// TIA Portal V16 export
// export: Created 2022-09-01T14:26:55.8686104Z, ExportSetting WithDefaults, DisplayName Totally Integrated Automation Portal, DisplayVersion V16, DisplayName TIA Portal Version Control Interface, DisplayVersion V16, DisplayName TIA Portal Openness, DisplayVersion V16, DisplayName STEP 7 Professional, DisplayVersion V16, DisplayName STEP 7 Safety, DisplayVersion V16, DisplayName WinCC Advanced, DisplayVersion V16
FUNCTION "Ciclo_Limpeza" : Void   // FC1, LAD
TITLE = Ciclo de lavagem e enxaguamento
{ S7_Optimized_Access := 'TRUE' }
VERSION : 0.1
// stored: AutoNumber true, IsIECCheckEnabled false, SetENOAutomatically false, UDAEnableTagReadback false
   VAR_TEMP   // added for the SCL form of the ladder/FBD networks
      _w1 : Bool;
      _w2 : Bool;
      _w3 : Bool;
   END_VAR
BEGIN

REGION Network 1: Etapa 1 (Início)
   // Início com EV's na posição de filtração. As bombas podem estar ligadas ou não, conforme a posição do switch 4
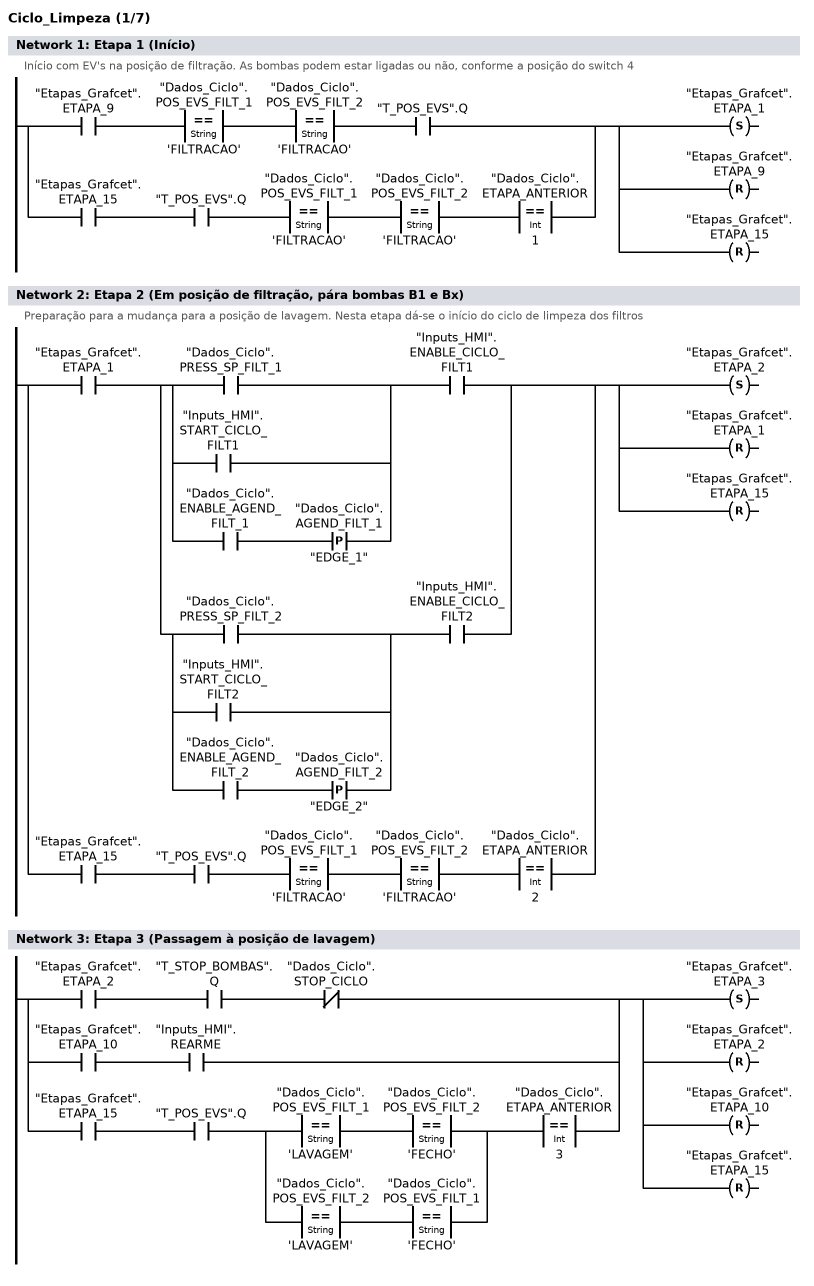
   RUNG wire#powerrail
      Contact( "Etapas_Grafcet".ETAPA_9 )
      { S7_Templates := "SrcType := String" } EQ_Contact(in1 := "Dados_Ciclo".POS_EVS_FILT_1, in2 := 'FILTRACAO')
      { S7_Templates := "SrcType := String" } EQ_Contact(in1 := "Dados_Ciclo".POS_EVS_FILT_2, in2 := 'FILTRACAO')
      Contact( "T_POS_EVS".Q )
      wire#w1
      S_Coil( "Etapas_Grafcet".ETAPA_1 )
   END_RUNG
   RUNG wire#powerrail
      Contact( "Etapas_Grafcet".ETAPA_15 )
      Contact( "T_POS_EVS".Q )
      { S7_Templates := "SrcType := String" } EQ_Contact(in1 := "Dados_Ciclo".POS_EVS_FILT_1, in2 := 'FILTRACAO')
      { S7_Templates := "SrcType := String" } EQ_Contact(in1 := "Dados_Ciclo".POS_EVS_FILT_2, in2 := 'FILTRACAO')
      { S7_Templates := "SrcType := Int" } EQ_Contact(in1 := "Dados_Ciclo".ETAPA_ANTERIOR, in2 := 1)
   END_RUNG wire#w1
   RUNG wire#w1
      R_Coil( "Etapas_Grafcet".ETAPA_9 )
   END_RUNG
   RUNG wire#w1
      R_Coil( "Etapas_Grafcet".ETAPA_15 )
   END_RUNG
   // the same network as SCL:
   IF ("Etapas_Grafcet".ETAPA_9 AND ("Dados_Ciclo".POS_EVS_FILT_1 = 'FILTRACAO') AND ("Dados_Ciclo".POS_EVS_FILT_2 = 'FILTRACAO') AND "T_POS_EVS".Q) OR ("Etapas_Grafcet".ETAPA_15 AND "T_POS_EVS".Q AND ("Dados_Ciclo".POS_EVS_FILT_1 = 'FILTRACAO') AND ("Dados_Ciclo".POS_EVS_FILT_2 = 'FILTRACAO') AND ("Dados_Ciclo".ETAPA_ANTERIOR = 1)) THEN
       "Etapas_Grafcet".ETAPA_1 := TRUE;
   END_IF;
   #_w1 := ("Etapas_Grafcet".ETAPA_9 AND ("Dados_Ciclo".POS_EVS_FILT_1 = 'FILTRACAO') AND ("Dados_Ciclo".POS_EVS_FILT_2 = 'FILTRACAO') AND "T_POS_EVS".Q) OR ("Etapas_Grafcet".ETAPA_15 AND "T_POS_EVS".Q AND ("Dados_Ciclo".POS_EVS_FILT_1 = 'FILTRACAO') AND ("Dados_Ciclo".POS_EVS_FILT_2 = 'FILTRACAO') AND ("Dados_Ciclo".ETAPA_ANTERIOR = 1));
   IF #_w1 THEN
       "Etapas_Grafcet".ETAPA_9 := FALSE;
       "Etapas_Grafcet".ETAPA_15 := FALSE;
   END_IF;
END_REGION

REGION Network 2: Etapa 2 (Em posição de filtração, pára bombas B1 e Bx)
   // Preparação para a mudança para a posição de lavagem. Nesta etapa dá-se o início do ciclo de limpeza dos filtros
   RUNG wire#powerrail
      Contact( "Etapas_Grafcet".ETAPA_1 )
      wire#w1
      Contact( "Dados_Ciclo".PRESS_SP_FILT_1 )
      wire#w2
      Contact( "Inputs_HMI".ENABLE_CICLO_FILT1 )
      wire#w3
      S_Coil( "Etapas_Grafcet".ETAPA_2 )
   END_RUNG
   RUNG wire#w1
      Contact( "Inputs_HMI".START_CICLO_FILT1 )
   END_RUNG wire#w2
   RUNG wire#w1
      Contact( "Dados_Ciclo".ENABLE_AGEND_FILT_1 )
      P_Contact(operand := "Dados_Ciclo".AGEND_FILT_1, bit := "EDGE_1")
   END_RUNG wire#w2
   RUNG wire#w1
      Contact( "Dados_Ciclo".PRESS_SP_FILT_2 )
      wire#w4
      Contact( "Inputs_HMI".ENABLE_CICLO_FILT2 )
   END_RUNG wire#w3
   RUNG wire#w1
      Contact( "Inputs_HMI".START_CICLO_FILT2 )
   END_RUNG wire#w4
   RUNG wire#w1
      Contact( "Dados_Ciclo".ENABLE_AGEND_FILT_2 )
      P_Contact(operand := "Dados_Ciclo".AGEND_FILT_2, bit := "EDGE_2")
   END_RUNG wire#w4
   RUNG wire#powerrail
      Contact( "Etapas_Grafcet".ETAPA_15 )
      Contact( "T_POS_EVS".Q )
      { S7_Templates := "SrcType := String" } EQ_Contact(in1 := "Dados_Ciclo".POS_EVS_FILT_1, in2 := 'FILTRACAO')
      { S7_Templates := "SrcType := String" } EQ_Contact(in1 := "Dados_Ciclo".POS_EVS_FILT_2, in2 := 'FILTRACAO')
      { S7_Templates := "SrcType := Int" } EQ_Contact(in1 := "Dados_Ciclo".ETAPA_ANTERIOR, in2 := 2)
   END_RUNG wire#w3
   RUNG wire#w3
      R_Coil( "Etapas_Grafcet".ETAPA_1 )
   END_RUNG
   RUNG wire#w3
      R_Coil( "Etapas_Grafcet".ETAPA_15 )
   END_RUNG
   // the same network as SCL:
   #_w1 := "Etapas_Grafcet".ETAPA_1 AND "Dados_Ciclo".ENABLE_AGEND_FILT_1 AND "Dados_Ciclo".AGEND_FILT_1 AND NOT "EDGE_1";   // rising edge of "Dados_Ciclo".AGEND_FILT_1
   "EDGE_1" := "Dados_Ciclo".AGEND_FILT_1;
   #_w2 := "Etapas_Grafcet".ETAPA_1 AND "Dados_Ciclo".ENABLE_AGEND_FILT_2 AND "Dados_Ciclo".AGEND_FILT_2 AND NOT "EDGE_2";   // rising edge of "Dados_Ciclo".AGEND_FILT_2
   "EDGE_2" := "Dados_Ciclo".AGEND_FILT_2;
   IF ((("Etapas_Grafcet".ETAPA_1 AND ("Dados_Ciclo".PRESS_SP_FILT_1 OR "Inputs_HMI".START_CICLO_FILT1)) OR #_w1) AND "Inputs_HMI".ENABLE_CICLO_FILT1) OR ((("Etapas_Grafcet".ETAPA_1 AND ("Dados_Ciclo".PRESS_SP_FILT_2 OR "Inputs_HMI".START_CICLO_FILT2)) OR #_w2) AND "Inputs_HMI".ENABLE_CICLO_FILT2) OR ("Etapas_Grafcet".ETAPA_15 AND "T_POS_EVS".Q AND ("Dados_Ciclo".POS_EVS_FILT_1 = 'FILTRACAO') AND ("Dados_Ciclo".POS_EVS_FILT_2 = 'FILTRACAO') AND ("Dados_Ciclo".ETAPA_ANTERIOR = 2)) THEN
       "Etapas_Grafcet".ETAPA_2 := TRUE;
   END_IF;
   #_w3 := ((("Etapas_Grafcet".ETAPA_1 AND ("Dados_Ciclo".PRESS_SP_FILT_1 OR "Inputs_HMI".START_CICLO_FILT1)) OR #_w1) AND "Inputs_HMI".ENABLE_CICLO_FILT1) OR ((("Etapas_Grafcet".ETAPA_1 AND ("Dados_Ciclo".PRESS_SP_FILT_2 OR "Inputs_HMI".START_CICLO_FILT2)) OR #_w2) AND "Inputs_HMI".ENABLE_CICLO_FILT2) OR ("Etapas_Grafcet".ETAPA_15 AND "T_POS_EVS".Q AND ("Dados_Ciclo".POS_EVS_FILT_1 = 'FILTRACAO') AND ("Dados_Ciclo".POS_EVS_FILT_2 = 'FILTRACAO') AND ("Dados_Ciclo".ETAPA_ANTERIOR = 2));
   IF #_w3 THEN
       "Etapas_Grafcet".ETAPA_1 := FALSE;
       "Etapas_Grafcet".ETAPA_15 := FALSE;
   END_IF;
END_REGION

REGION Network 3: Etapa 3 (Passagem à posição de lavagem)
   RUNG wire#powerrail
      Contact( "Etapas_Grafcet".ETAPA_2 )
      Contact( "T_STOP_BOMBAS".Q )
      I_Contact( "Dados_Ciclo".STOP_CICLO )
      wire#w1
      S_Coil( "Etapas_Grafcet".ETAPA_3 )
   END_RUNG
   RUNG wire#powerrail
      Contact( "Etapas_Grafcet".ETAPA_10 )
      Contact( "Inputs_HMI".REARME )
   END_RUNG wire#w1
   RUNG wire#powerrail
      Contact( "Etapas_Grafcet".ETAPA_15 )
      Contact( "T_POS_EVS".Q )
      wire#w2
      { S7_Templates := "SrcType := String" } EQ_Contact(in1 := "Dados_Ciclo".POS_EVS_FILT_1, in2 := 'LAVAGEM')
      { S7_Templates := "SrcType := String" } EQ_Contact(in1 := "Dados_Ciclo".POS_EVS_FILT_2, in2 := 'FECHO')
      wire#w3
      { S7_Templates := "SrcType := Int" } EQ_Contact(in1 := "Dados_Ciclo".ETAPA_ANTERIOR, in2 := 3)
   END_RUNG wire#w1
   RUNG wire#w2
      { S7_Templates := "SrcType := String" } EQ_Contact(in1 := "Dados_Ciclo".POS_EVS_FILT_2, in2 := 'LAVAGEM')
      { S7_Templates := "SrcType := String" } EQ_Contact(in1 := "Dados_Ciclo".POS_EVS_FILT_1, in2 := 'FECHO')
   END_RUNG wire#w3
   RUNG wire#w1
      R_Coil( "Etapas_Grafcet".ETAPA_2 )
   END_RUNG
   RUNG wire#w1
      R_Coil( "Etapas_Grafcet".ETAPA_10 )
   END_RUNG
   RUNG wire#w1
      R_Coil( "Etapas_Grafcet".ETAPA_15 )
   END_RUNG
   // the same network as SCL:
   IF ("Etapas_Grafcet".ETAPA_2 AND "T_STOP_BOMBAS".Q AND NOT "Dados_Ciclo".STOP_CICLO) OR ("Etapas_Grafcet".ETAPA_10 AND "Inputs_HMI".REARME) OR ("Etapas_Grafcet".ETAPA_15 AND "T_POS_EVS".Q AND ((("Dados_Ciclo".POS_EVS_FILT_1 = 'LAVAGEM') AND ("Dados_Ciclo".POS_EVS_FILT_2 = 'FECHO')) OR (("Dados_Ciclo".POS_EVS_FILT_2 = 'LAVAGEM') AND ("Dados_Ciclo".POS_EVS_FILT_1 = 'FECHO'))) AND ("Dados_Ciclo".ETAPA_ANTERIOR = 3)) THEN
       "Etapas_Grafcet".ETAPA_3 := TRUE;
   END_IF;
   #_w1 := ("Etapas_Grafcet".ETAPA_2 AND "T_STOP_BOMBAS".Q AND NOT "Dados_Ciclo".STOP_CICLO) OR ("Etapas_Grafcet".ETAPA_10 AND "Inputs_HMI".REARME) OR ("Etapas_Grafcet".ETAPA_15 AND "T_POS_EVS".Q AND ((("Dados_Ciclo".POS_EVS_FILT_1 = 'LAVAGEM') AND ("Dados_Ciclo".POS_EVS_FILT_2 = 'FECHO')) OR (("Dados_Ciclo".POS_EVS_FILT_2 = 'LAVAGEM') AND ("Dados_Ciclo".POS_EVS_FILT_1 = 'FECHO'))) AND ("Dados_Ciclo".ETAPA_ANTERIOR = 3));
   IF #_w1 THEN
       "Etapas_Grafcet".ETAPA_2 := FALSE;
       "Etapas_Grafcet".ETAPA_10 := FALSE;
       "Etapas_Grafcet".ETAPA_15 := FALSE;
   END_IF;
END_REGION

REGION Network 4: Etapa 4 (Em lavagem, B1 e BX ligadas)
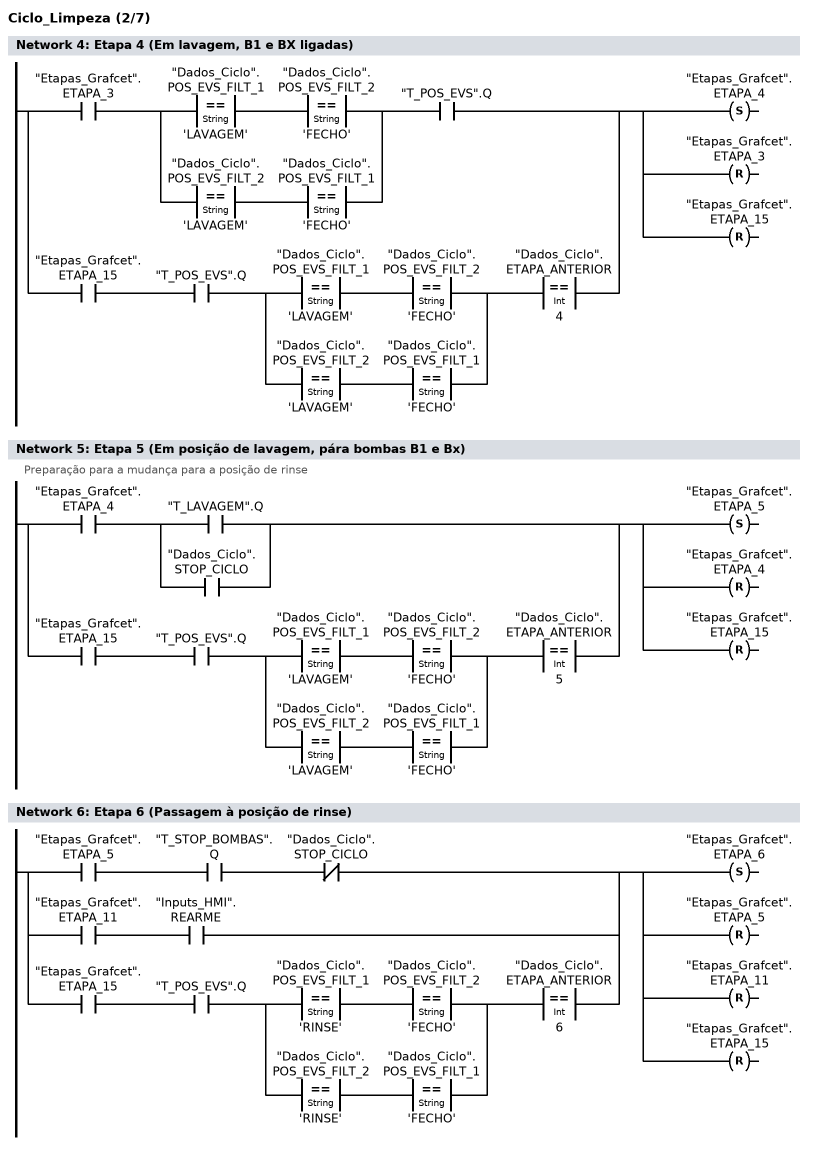
   RUNG wire#powerrail
      Contact( "Etapas_Grafcet".ETAPA_3 )
      wire#w1
      { S7_Templates := "SrcType := String" } EQ_Contact(in1 := "Dados_Ciclo".POS_EVS_FILT_1, in2 := 'LAVAGEM')
      { S7_Templates := "SrcType := String" } EQ_Contact(in1 := "Dados_Ciclo".POS_EVS_FILT_2, in2 := 'FECHO')
      wire#w2
      Contact( "T_POS_EVS".Q )
      wire#w3
      S_Coil( "Etapas_Grafcet".ETAPA_4 )
   END_RUNG
   RUNG wire#w1
      { S7_Templates := "SrcType := String" } EQ_Contact(in1 := "Dados_Ciclo".POS_EVS_FILT_2, in2 := 'LAVAGEM')
      { S7_Templates := "SrcType := String" } EQ_Contact(in1 := "Dados_Ciclo".POS_EVS_FILT_1, in2 := 'FECHO')
   END_RUNG wire#w2
   RUNG wire#powerrail
      Contact( "Etapas_Grafcet".ETAPA_15 )
      Contact( "T_POS_EVS".Q )
      wire#w4
      { S7_Templates := "SrcType := String" } EQ_Contact(in1 := "Dados_Ciclo".POS_EVS_FILT_1, in2 := 'LAVAGEM')
      { S7_Templates := "SrcType := String" } EQ_Contact(in1 := "Dados_Ciclo".POS_EVS_FILT_2, in2 := 'FECHO')
      wire#w5
      { S7_Templates := "SrcType := Int" } EQ_Contact(in1 := "Dados_Ciclo".ETAPA_ANTERIOR, in2 := 4)
   END_RUNG wire#w3
   RUNG wire#w4
      { S7_Templates := "SrcType := String" } EQ_Contact(in1 := "Dados_Ciclo".POS_EVS_FILT_2, in2 := 'LAVAGEM')
      { S7_Templates := "SrcType := String" } EQ_Contact(in1 := "Dados_Ciclo".POS_EVS_FILT_1, in2 := 'FECHO')
   END_RUNG wire#w5
   RUNG wire#w3
      R_Coil( "Etapas_Grafcet".ETAPA_3 )
   END_RUNG
   RUNG wire#w3
      R_Coil( "Etapas_Grafcet".ETAPA_15 )
   END_RUNG
   // the same network as SCL:
   IF ("Etapas_Grafcet".ETAPA_3 AND ((("Dados_Ciclo".POS_EVS_FILT_1 = 'LAVAGEM') AND ("Dados_Ciclo".POS_EVS_FILT_2 = 'FECHO')) OR (("Dados_Ciclo".POS_EVS_FILT_2 = 'LAVAGEM') AND ("Dados_Ciclo".POS_EVS_FILT_1 = 'FECHO'))) AND "T_POS_EVS".Q) OR ("Etapas_Grafcet".ETAPA_15 AND "T_POS_EVS".Q AND ((("Dados_Ciclo".POS_EVS_FILT_1 = 'LAVAGEM') AND ("Dados_Ciclo".POS_EVS_FILT_2 = 'FECHO')) OR (("Dados_Ciclo".POS_EVS_FILT_2 = 'LAVAGEM') AND ("Dados_Ciclo".POS_EVS_FILT_1 = 'FECHO'))) AND ("Dados_Ciclo".ETAPA_ANTERIOR = 4)) THEN
       "Etapas_Grafcet".ETAPA_4 := TRUE;
   END_IF;
   #_w1 := ("Etapas_Grafcet".ETAPA_3 AND ((("Dados_Ciclo".POS_EVS_FILT_1 = 'LAVAGEM') AND ("Dados_Ciclo".POS_EVS_FILT_2 = 'FECHO')) OR (("Dados_Ciclo".POS_EVS_FILT_2 = 'LAVAGEM') AND ("Dados_Ciclo".POS_EVS_FILT_1 = 'FECHO'))) AND "T_POS_EVS".Q) OR ("Etapas_Grafcet".ETAPA_15 AND "T_POS_EVS".Q AND ((("Dados_Ciclo".POS_EVS_FILT_1 = 'LAVAGEM') AND ("Dados_Ciclo".POS_EVS_FILT_2 = 'FECHO')) OR (("Dados_Ciclo".POS_EVS_FILT_2 = 'LAVAGEM') AND ("Dados_Ciclo".POS_EVS_FILT_1 = 'FECHO'))) AND ("Dados_Ciclo".ETAPA_ANTERIOR = 4));
   IF #_w1 THEN
       "Etapas_Grafcet".ETAPA_3 := FALSE;
       "Etapas_Grafcet".ETAPA_15 := FALSE;
   END_IF;
END_REGION

REGION Network 5: Etapa 5 (Em posição de lavagem, pára bombas B1 e Bx)
   // Preparação para a mudança para a posição de rinse
   RUNG wire#powerrail
      Contact( "Etapas_Grafcet".ETAPA_4 )
      wire#w1
      Contact( "T_LAVAGEM".Q )
      wire#w2
      S_Coil( "Etapas_Grafcet".ETAPA_5 )
   END_RUNG
   RUNG wire#w1
      Contact( "Dados_Ciclo".STOP_CICLO )
   END_RUNG wire#w2
   RUNG wire#powerrail
      Contact( "Etapas_Grafcet".ETAPA_15 )
      Contact( "T_POS_EVS".Q )
      wire#w3
      { S7_Templates := "SrcType := String" } EQ_Contact(in1 := "Dados_Ciclo".POS_EVS_FILT_1, in2 := 'LAVAGEM')
      { S7_Templates := "SrcType := String" } EQ_Contact(in1 := "Dados_Ciclo".POS_EVS_FILT_2, in2 := 'FECHO')
      wire#w4
      { S7_Templates := "SrcType := Int" } EQ_Contact(in1 := "Dados_Ciclo".ETAPA_ANTERIOR, in2 := 5)
   END_RUNG wire#w2
   RUNG wire#w3
      { S7_Templates := "SrcType := String" } EQ_Contact(in1 := "Dados_Ciclo".POS_EVS_FILT_2, in2 := 'LAVAGEM')
      { S7_Templates := "SrcType := String" } EQ_Contact(in1 := "Dados_Ciclo".POS_EVS_FILT_1, in2 := 'FECHO')
   END_RUNG wire#w4
   RUNG wire#w2
      R_Coil( "Etapas_Grafcet".ETAPA_4 )
   END_RUNG
   RUNG wire#w2
      R_Coil( "Etapas_Grafcet".ETAPA_15 )
   END_RUNG
   // the same network as SCL:
   IF ("Etapas_Grafcet".ETAPA_4 AND ("T_LAVAGEM".Q OR "Dados_Ciclo".STOP_CICLO)) OR ("Etapas_Grafcet".ETAPA_15 AND "T_POS_EVS".Q AND ((("Dados_Ciclo".POS_EVS_FILT_1 = 'LAVAGEM') AND ("Dados_Ciclo".POS_EVS_FILT_2 = 'FECHO')) OR (("Dados_Ciclo".POS_EVS_FILT_2 = 'LAVAGEM') AND ("Dados_Ciclo".POS_EVS_FILT_1 = 'FECHO'))) AND ("Dados_Ciclo".ETAPA_ANTERIOR = 5)) THEN
       "Etapas_Grafcet".ETAPA_5 := TRUE;
   END_IF;
   #_w1 := ("Etapas_Grafcet".ETAPA_4 AND ("T_LAVAGEM".Q OR "Dados_Ciclo".STOP_CICLO)) OR ("Etapas_Grafcet".ETAPA_15 AND "T_POS_EVS".Q AND ((("Dados_Ciclo".POS_EVS_FILT_1 = 'LAVAGEM') AND ("Dados_Ciclo".POS_EVS_FILT_2 = 'FECHO')) OR (("Dados_Ciclo".POS_EVS_FILT_2 = 'LAVAGEM') AND ("Dados_Ciclo".POS_EVS_FILT_1 = 'FECHO'))) AND ("Dados_Ciclo".ETAPA_ANTERIOR = 5));
   IF #_w1 THEN
       "Etapas_Grafcet".ETAPA_4 := FALSE;
       "Etapas_Grafcet".ETAPA_15 := FALSE;
   END_IF;
END_REGION

REGION Network 6: Etapa 6 (Passagem à posição de rinse)
   RUNG wire#powerrail
      Contact( "Etapas_Grafcet".ETAPA_5 )
      Contact( "T_STOP_BOMBAS".Q )
      I_Contact( "Dados_Ciclo".STOP_CICLO )
      wire#w1
      S_Coil( "Etapas_Grafcet".ETAPA_6 )
   END_RUNG
   RUNG wire#powerrail
      Contact( "Etapas_Grafcet".ETAPA_11 )
      Contact( "Inputs_HMI".REARME )
   END_RUNG wire#w1
   RUNG wire#powerrail
      Contact( "Etapas_Grafcet".ETAPA_15 )
      Contact( "T_POS_EVS".Q )
      wire#w2
      { S7_Templates := "SrcType := String" } EQ_Contact(in1 := "Dados_Ciclo".POS_EVS_FILT_1, in2 := 'RINSE')
      { S7_Templates := "SrcType := String" } EQ_Contact(in1 := "Dados_Ciclo".POS_EVS_FILT_2, in2 := 'FECHO')
      wire#w3
      { S7_Templates := "SrcType := Int" } EQ_Contact(in1 := "Dados_Ciclo".ETAPA_ANTERIOR, in2 := 6)
   END_RUNG wire#w1
   RUNG wire#w2
      { S7_Templates := "SrcType := String" } EQ_Contact(in1 := "Dados_Ciclo".POS_EVS_FILT_2, in2 := 'RINSE')
      { S7_Templates := "SrcType := String" } EQ_Contact(in1 := "Dados_Ciclo".POS_EVS_FILT_1, in2 := 'FECHO')
   END_RUNG wire#w3
   RUNG wire#w1
      R_Coil( "Etapas_Grafcet".ETAPA_5 )
   END_RUNG
   RUNG wire#w1
      R_Coil( "Etapas_Grafcet".ETAPA_11 )
   END_RUNG
   RUNG wire#w1
      R_Coil( "Etapas_Grafcet".ETAPA_15 )
   END_RUNG
   // the same network as SCL:
   IF ("Etapas_Grafcet".ETAPA_5 AND "T_STOP_BOMBAS".Q AND NOT "Dados_Ciclo".STOP_CICLO) OR ("Etapas_Grafcet".ETAPA_11 AND "Inputs_HMI".REARME) OR ("Etapas_Grafcet".ETAPA_15 AND "T_POS_EVS".Q AND ((("Dados_Ciclo".POS_EVS_FILT_1 = 'RINSE') AND ("Dados_Ciclo".POS_EVS_FILT_2 = 'FECHO')) OR (("Dados_Ciclo".POS_EVS_FILT_2 = 'RINSE') AND ("Dados_Ciclo".POS_EVS_FILT_1 = 'FECHO'))) AND ("Dados_Ciclo".ETAPA_ANTERIOR = 6)) THEN
       "Etapas_Grafcet".ETAPA_6 := TRUE;
   END_IF;
   #_w1 := ("Etapas_Grafcet".ETAPA_5 AND "T_STOP_BOMBAS".Q AND NOT "Dados_Ciclo".STOP_CICLO) OR ("Etapas_Grafcet".ETAPA_11 AND "Inputs_HMI".REARME) OR ("Etapas_Grafcet".ETAPA_15 AND "T_POS_EVS".Q AND ((("Dados_Ciclo".POS_EVS_FILT_1 = 'RINSE') AND ("Dados_Ciclo".POS_EVS_FILT_2 = 'FECHO')) OR (("Dados_Ciclo".POS_EVS_FILT_2 = 'RINSE') AND ("Dados_Ciclo".POS_EVS_FILT_1 = 'FECHO'))) AND ("Dados_Ciclo".ETAPA_ANTERIOR = 6));
   IF #_w1 THEN
       "Etapas_Grafcet".ETAPA_5 := FALSE;
       "Etapas_Grafcet".ETAPA_11 := FALSE;
       "Etapas_Grafcet".ETAPA_15 := FALSE;
   END_IF;
END_REGION

REGION Network 7: Etapa 7 (Em rinse, B1 ligada)
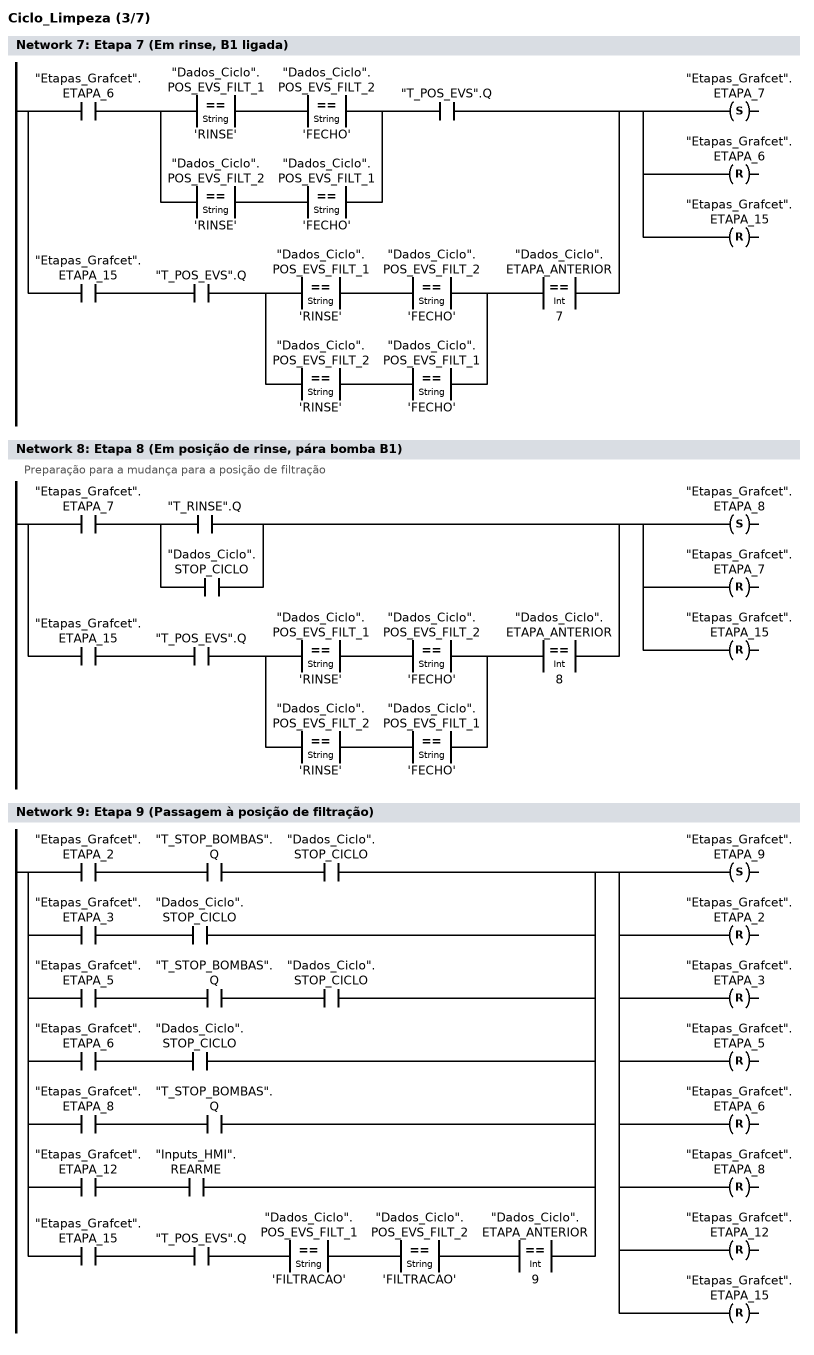
   RUNG wire#powerrail
      Contact( "Etapas_Grafcet".ETAPA_6 )
      wire#w1
      { S7_Templates := "SrcType := String" } EQ_Contact(in1 := "Dados_Ciclo".POS_EVS_FILT_1, in2 := 'RINSE')
      { S7_Templates := "SrcType := String" } EQ_Contact(in1 := "Dados_Ciclo".POS_EVS_FILT_2, in2 := 'FECHO')
      wire#w2
      Contact( "T_POS_EVS".Q )
      wire#w3
      S_Coil( "Etapas_Grafcet".ETAPA_7 )
   END_RUNG
   RUNG wire#w1
      { S7_Templates := "SrcType := String" } EQ_Contact(in1 := "Dados_Ciclo".POS_EVS_FILT_2, in2 := 'RINSE')
      { S7_Templates := "SrcType := String" } EQ_Contact(in1 := "Dados_Ciclo".POS_EVS_FILT_1, in2 := 'FECHO')
   END_RUNG wire#w2
   RUNG wire#powerrail
      Contact( "Etapas_Grafcet".ETAPA_15 )
      Contact( "T_POS_EVS".Q )
      wire#w4
      { S7_Templates := "SrcType := String" } EQ_Contact(in1 := "Dados_Ciclo".POS_EVS_FILT_1, in2 := 'RINSE')
      { S7_Templates := "SrcType := String" } EQ_Contact(in1 := "Dados_Ciclo".POS_EVS_FILT_2, in2 := 'FECHO')
      wire#w5
      { S7_Templates := "SrcType := Int" } EQ_Contact(in1 := "Dados_Ciclo".ETAPA_ANTERIOR, in2 := 7)
   END_RUNG wire#w3
   RUNG wire#w4
      { S7_Templates := "SrcType := String" } EQ_Contact(in1 := "Dados_Ciclo".POS_EVS_FILT_2, in2 := 'RINSE')
      { S7_Templates := "SrcType := String" } EQ_Contact(in1 := "Dados_Ciclo".POS_EVS_FILT_1, in2 := 'FECHO')
   END_RUNG wire#w5
   RUNG wire#w3
      R_Coil( "Etapas_Grafcet".ETAPA_6 )
   END_RUNG
   RUNG wire#w3
      R_Coil( "Etapas_Grafcet".ETAPA_15 )
   END_RUNG
   // the same network as SCL:
   IF ("Etapas_Grafcet".ETAPA_6 AND ((("Dados_Ciclo".POS_EVS_FILT_1 = 'RINSE') AND ("Dados_Ciclo".POS_EVS_FILT_2 = 'FECHO')) OR (("Dados_Ciclo".POS_EVS_FILT_2 = 'RINSE') AND ("Dados_Ciclo".POS_EVS_FILT_1 = 'FECHO'))) AND "T_POS_EVS".Q) OR ("Etapas_Grafcet".ETAPA_15 AND "T_POS_EVS".Q AND ((("Dados_Ciclo".POS_EVS_FILT_1 = 'RINSE') AND ("Dados_Ciclo".POS_EVS_FILT_2 = 'FECHO')) OR (("Dados_Ciclo".POS_EVS_FILT_2 = 'RINSE') AND ("Dados_Ciclo".POS_EVS_FILT_1 = 'FECHO'))) AND ("Dados_Ciclo".ETAPA_ANTERIOR = 7)) THEN
       "Etapas_Grafcet".ETAPA_7 := TRUE;
   END_IF;
   #_w1 := ("Etapas_Grafcet".ETAPA_6 AND ((("Dados_Ciclo".POS_EVS_FILT_1 = 'RINSE') AND ("Dados_Ciclo".POS_EVS_FILT_2 = 'FECHO')) OR (("Dados_Ciclo".POS_EVS_FILT_2 = 'RINSE') AND ("Dados_Ciclo".POS_EVS_FILT_1 = 'FECHO'))) AND "T_POS_EVS".Q) OR ("Etapas_Grafcet".ETAPA_15 AND "T_POS_EVS".Q AND ((("Dados_Ciclo".POS_EVS_FILT_1 = 'RINSE') AND ("Dados_Ciclo".POS_EVS_FILT_2 = 'FECHO')) OR (("Dados_Ciclo".POS_EVS_FILT_2 = 'RINSE') AND ("Dados_Ciclo".POS_EVS_FILT_1 = 'FECHO'))) AND ("Dados_Ciclo".ETAPA_ANTERIOR = 7));
   IF #_w1 THEN
       "Etapas_Grafcet".ETAPA_6 := FALSE;
       "Etapas_Grafcet".ETAPA_15 := FALSE;
   END_IF;
END_REGION

REGION Network 8: Etapa 8 (Em posição de rinse, pára bomba B1)
   // Preparação para a mudança para a posição de filtração
   RUNG wire#powerrail
      Contact( "Etapas_Grafcet".ETAPA_7 )
      wire#w1
      Contact( "T_RINSE".Q )
      wire#w2
      S_Coil( "Etapas_Grafcet".ETAPA_8 )
   END_RUNG
   RUNG wire#w1
      Contact( "Dados_Ciclo".STOP_CICLO )
   END_RUNG wire#w2
   RUNG wire#powerrail
      Contact( "Etapas_Grafcet".ETAPA_15 )
      Contact( "T_POS_EVS".Q )
      wire#w3
      { S7_Templates := "SrcType := String" } EQ_Contact(in1 := "Dados_Ciclo".POS_EVS_FILT_1, in2 := 'RINSE')
      { S7_Templates := "SrcType := String" } EQ_Contact(in1 := "Dados_Ciclo".POS_EVS_FILT_2, in2 := 'FECHO')
      wire#w4
      { S7_Templates := "SrcType := Int" } EQ_Contact(in1 := "Dados_Ciclo".ETAPA_ANTERIOR, in2 := 8)
   END_RUNG wire#w2
   RUNG wire#w3
      { S7_Templates := "SrcType := String" } EQ_Contact(in1 := "Dados_Ciclo".POS_EVS_FILT_2, in2 := 'RINSE')
      { S7_Templates := "SrcType := String" } EQ_Contact(in1 := "Dados_Ciclo".POS_EVS_FILT_1, in2 := 'FECHO')
   END_RUNG wire#w4
   RUNG wire#w2
      R_Coil( "Etapas_Grafcet".ETAPA_7 )
   END_RUNG
   RUNG wire#w2
      R_Coil( "Etapas_Grafcet".ETAPA_15 )
   END_RUNG
   // the same network as SCL:
   IF ("Etapas_Grafcet".ETAPA_7 AND ("T_RINSE".Q OR "Dados_Ciclo".STOP_CICLO)) OR ("Etapas_Grafcet".ETAPA_15 AND "T_POS_EVS".Q AND ((("Dados_Ciclo".POS_EVS_FILT_1 = 'RINSE') AND ("Dados_Ciclo".POS_EVS_FILT_2 = 'FECHO')) OR (("Dados_Ciclo".POS_EVS_FILT_2 = 'RINSE') AND ("Dados_Ciclo".POS_EVS_FILT_1 = 'FECHO'))) AND ("Dados_Ciclo".ETAPA_ANTERIOR = 8)) THEN
       "Etapas_Grafcet".ETAPA_8 := TRUE;
   END_IF;
   #_w1 := ("Etapas_Grafcet".ETAPA_7 AND ("T_RINSE".Q OR "Dados_Ciclo".STOP_CICLO)) OR ("Etapas_Grafcet".ETAPA_15 AND "T_POS_EVS".Q AND ((("Dados_Ciclo".POS_EVS_FILT_1 = 'RINSE') AND ("Dados_Ciclo".POS_EVS_FILT_2 = 'FECHO')) OR (("Dados_Ciclo".POS_EVS_FILT_2 = 'RINSE') AND ("Dados_Ciclo".POS_EVS_FILT_1 = 'FECHO'))) AND ("Dados_Ciclo".ETAPA_ANTERIOR = 8));
   IF #_w1 THEN
       "Etapas_Grafcet".ETAPA_7 := FALSE;
       "Etapas_Grafcet".ETAPA_15 := FALSE;
   END_IF;
END_REGION

REGION Network 9: Etapa 9 (Passagem à posição de filtração)
   RUNG wire#powerrail
      Contact( "Etapas_Grafcet".ETAPA_2 )
      Contact( "T_STOP_BOMBAS".Q )
      Contact( "Dados_Ciclo".STOP_CICLO )
      wire#w1
      S_Coil( "Etapas_Grafcet".ETAPA_9 )
   END_RUNG
   RUNG wire#powerrail
      Contact( "Etapas_Grafcet".ETAPA_3 )
      Contact( "Dados_Ciclo".STOP_CICLO )
   END_RUNG wire#w1
   RUNG wire#powerrail
      Contact( "Etapas_Grafcet".ETAPA_5 )
      Contact( "T_STOP_BOMBAS".Q )
      Contact( "Dados_Ciclo".STOP_CICLO )
   END_RUNG wire#w1
   RUNG wire#powerrail
      Contact( "Etapas_Grafcet".ETAPA_6 )
      Contact( "Dados_Ciclo".STOP_CICLO )
   END_RUNG wire#w1
   RUNG wire#powerrail
      Contact( "Etapas_Grafcet".ETAPA_8 )
      Contact( "T_STOP_BOMBAS".Q )
   END_RUNG wire#w1
   RUNG wire#powerrail
      Contact( "Etapas_Grafcet".ETAPA_12 )
      Contact( "Inputs_HMI".REARME )
   END_RUNG wire#w1
   RUNG wire#powerrail
      Contact( "Etapas_Grafcet".ETAPA_15 )
      Contact( "T_POS_EVS".Q )
      { S7_Templates := "SrcType := String" } EQ_Contact(in1 := "Dados_Ciclo".POS_EVS_FILT_1, in2 := 'FILTRACAO')
      { S7_Templates := "SrcType := String" } EQ_Contact(in1 := "Dados_Ciclo".POS_EVS_FILT_2, in2 := 'FILTRACAO')
      { S7_Templates := "SrcType := Int" } EQ_Contact(in1 := "Dados_Ciclo".ETAPA_ANTERIOR, in2 := 9)
   END_RUNG wire#w1
   RUNG wire#w1
      R_Coil( "Etapas_Grafcet".ETAPA_2 )
   END_RUNG
   RUNG wire#w1
      R_Coil( "Etapas_Grafcet".ETAPA_3 )
   END_RUNG
   RUNG wire#w1
      R_Coil( "Etapas_Grafcet".ETAPA_5 )
   END_RUNG
   RUNG wire#w1
      R_Coil( "Etapas_Grafcet".ETAPA_6 )
   END_RUNG
   RUNG wire#w1
      R_Coil( "Etapas_Grafcet".ETAPA_8 )
   END_RUNG
   RUNG wire#w1
      R_Coil( "Etapas_Grafcet".ETAPA_12 )
   END_RUNG
   RUNG wire#w1
      R_Coil( "Etapas_Grafcet".ETAPA_15 )
   END_RUNG
   // the same network as SCL:
   IF ("Etapas_Grafcet".ETAPA_2 AND "T_STOP_BOMBAS".Q AND "Dados_Ciclo".STOP_CICLO) OR ("Etapas_Grafcet".ETAPA_3 AND "Dados_Ciclo".STOP_CICLO) OR ("Etapas_Grafcet".ETAPA_5 AND "T_STOP_BOMBAS".Q AND "Dados_Ciclo".STOP_CICLO) OR ("Etapas_Grafcet".ETAPA_6 AND "Dados_Ciclo".STOP_CICLO) OR ("Etapas_Grafcet".ETAPA_8 AND "T_STOP_BOMBAS".Q) OR ("Etapas_Grafcet".ETAPA_12 AND "Inputs_HMI".REARME) OR ("Etapas_Grafcet".ETAPA_15 AND "T_POS_EVS".Q AND ("Dados_Ciclo".POS_EVS_FILT_1 = 'FILTRACAO') AND ("Dados_Ciclo".POS_EVS_FILT_2 = 'FILTRACAO') AND ("Dados_Ciclo".ETAPA_ANTERIOR = 9)) THEN
       "Etapas_Grafcet".ETAPA_9 := TRUE;
   END_IF;
   #_w1 := ("Etapas_Grafcet".ETAPA_2 AND "T_STOP_BOMBAS".Q AND "Dados_Ciclo".STOP_CICLO) OR ("Etapas_Grafcet".ETAPA_3 AND "Dados_Ciclo".STOP_CICLO) OR ("Etapas_Grafcet".ETAPA_5 AND "T_STOP_BOMBAS".Q AND "Dados_Ciclo".STOP_CICLO) OR ("Etapas_Grafcet".ETAPA_6 AND "Dados_Ciclo".STOP_CICLO) OR ("Etapas_Grafcet".ETAPA_8 AND "T_STOP_BOMBAS".Q) OR ("Etapas_Grafcet".ETAPA_12 AND "Inputs_HMI".REARME) OR ("Etapas_Grafcet".ETAPA_15 AND "T_POS_EVS".Q AND ("Dados_Ciclo".POS_EVS_FILT_1 = 'FILTRACAO') AND ("Dados_Ciclo".POS_EVS_FILT_2 = 'FILTRACAO') AND ("Dados_Ciclo".ETAPA_ANTERIOR = 9));
   IF #_w1 THEN
       "Etapas_Grafcet".ETAPA_2 := FALSE;
       "Etapas_Grafcet".ETAPA_3 := FALSE;
       "Etapas_Grafcet".ETAPA_5 := FALSE;
       "Etapas_Grafcet".ETAPA_6 := FALSE;
       "Etapas_Grafcet".ETAPA_8 := FALSE;
       "Etapas_Grafcet".ETAPA_12 := FALSE;
       "Etapas_Grafcet".ETAPA_15 := FALSE;
   END_IF;
END_REGION

REGION Network 10: ETAPA 10 (Alarme posição lavagem)
   // As ev's não estão na posição de lavagem / fecho
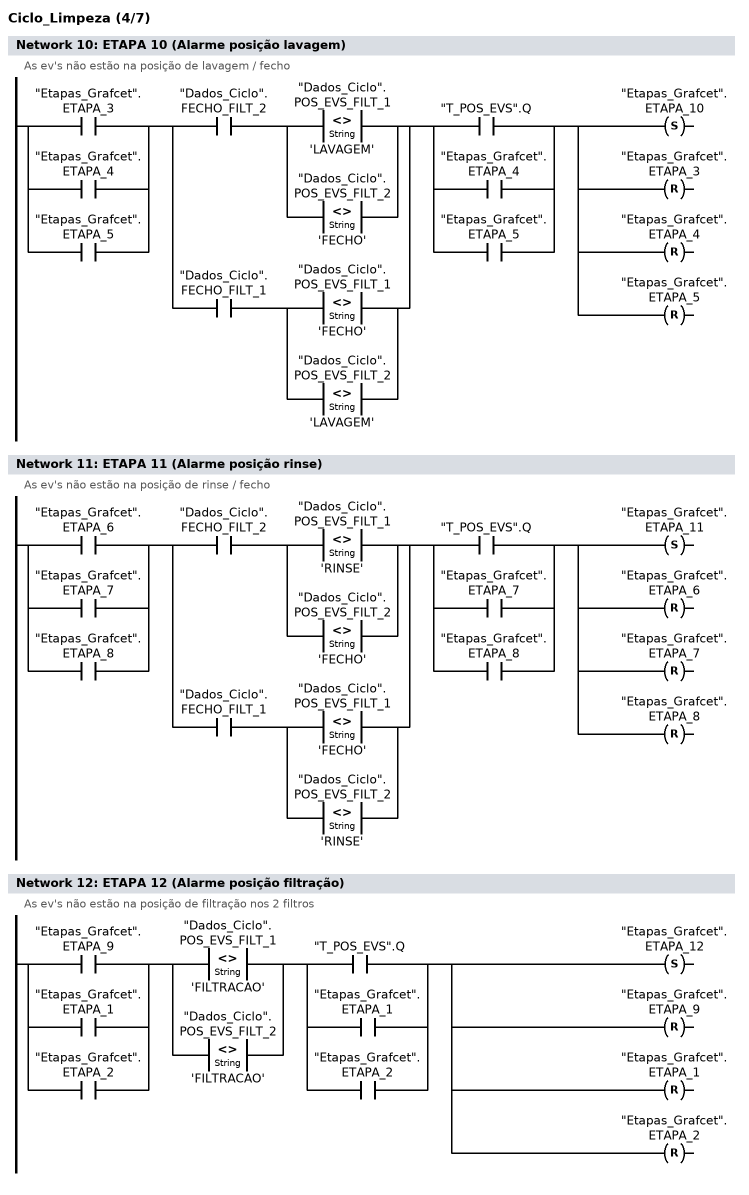
   RUNG wire#powerrail
      Contact( "Etapas_Grafcet".ETAPA_3 )
      wire#w1
      Contact( "Dados_Ciclo".FECHO_FILT_2 )
      wire#w2
      { S7_Templates := "SrcType := String" } NE_Contact(in1 := "Dados_Ciclo".POS_EVS_FILT_1, in2 := 'LAVAGEM')
      wire#w3
      Contact( "T_POS_EVS".Q )
      wire#w5
      S_Coil( "Etapas_Grafcet".ETAPA_10 )
   END_RUNG
   RUNG wire#powerrail
      Contact( "Etapas_Grafcet".ETAPA_4 )
   END_RUNG wire#w1
   RUNG wire#powerrail
      Contact( "Etapas_Grafcet".ETAPA_5 )
   END_RUNG wire#w1
   RUNG wire#w2
      { S7_Templates := "SrcType := String" } NE_Contact(in1 := "Dados_Ciclo".POS_EVS_FILT_2, in2 := 'FECHO')
   END_RUNG wire#w3
   RUNG wire#w1
      Contact( "Dados_Ciclo".FECHO_FILT_1 )
      wire#w4
      { S7_Templates := "SrcType := String" } NE_Contact(in1 := "Dados_Ciclo".POS_EVS_FILT_1, in2 := 'FECHO')
   END_RUNG wire#w3
   RUNG wire#w4
      { S7_Templates := "SrcType := String" } NE_Contact(in1 := "Dados_Ciclo".POS_EVS_FILT_2, in2 := 'LAVAGEM')
   END_RUNG wire#w3
   RUNG wire#w3
      Contact( "Etapas_Grafcet".ETAPA_4 )
   END_RUNG wire#w5
   RUNG wire#w3
      Contact( "Etapas_Grafcet".ETAPA_5 )
   END_RUNG wire#w5
   RUNG wire#w5
      R_Coil( "Etapas_Grafcet".ETAPA_3 )
   END_RUNG
   RUNG wire#w5
      R_Coil( "Etapas_Grafcet".ETAPA_4 )
   END_RUNG
   RUNG wire#w5
      R_Coil( "Etapas_Grafcet".ETAPA_5 )
   END_RUNG
   // the same network as SCL:
   IF ("Etapas_Grafcet".ETAPA_3 OR "Etapas_Grafcet".ETAPA_4 OR "Etapas_Grafcet".ETAPA_5) AND (("Dados_Ciclo".FECHO_FILT_2 AND (("Dados_Ciclo".POS_EVS_FILT_1 <> 'LAVAGEM') OR ("Dados_Ciclo".POS_EVS_FILT_2 <> 'FECHO'))) OR ("Dados_Ciclo".FECHO_FILT_1 AND (("Dados_Ciclo".POS_EVS_FILT_1 <> 'FECHO') OR ("Dados_Ciclo".POS_EVS_FILT_2 <> 'LAVAGEM')))) AND ("T_POS_EVS".Q OR "Etapas_Grafcet".ETAPA_4 OR "Etapas_Grafcet".ETAPA_5) THEN
       "Etapas_Grafcet".ETAPA_10 := TRUE;
   END_IF;
   #_w1 := ("Etapas_Grafcet".ETAPA_3 OR "Etapas_Grafcet".ETAPA_4 OR "Etapas_Grafcet".ETAPA_5) AND (("Dados_Ciclo".FECHO_FILT_2 AND (("Dados_Ciclo".POS_EVS_FILT_1 <> 'LAVAGEM') OR ("Dados_Ciclo".POS_EVS_FILT_2 <> 'FECHO'))) OR ("Dados_Ciclo".FECHO_FILT_1 AND (("Dados_Ciclo".POS_EVS_FILT_1 <> 'FECHO') OR ("Dados_Ciclo".POS_EVS_FILT_2 <> 'LAVAGEM')))) AND ("T_POS_EVS".Q OR "Etapas_Grafcet".ETAPA_4 OR "Etapas_Grafcet".ETAPA_5);
   IF #_w1 THEN
       "Etapas_Grafcet".ETAPA_3 := FALSE;
       "Etapas_Grafcet".ETAPA_4 := FALSE;
       "Etapas_Grafcet".ETAPA_5 := FALSE;
   END_IF;
END_REGION

REGION Network 11: ETAPA 11 (Alarme posição rinse)
   // As ev's não estão na posição de rinse / fecho
   RUNG wire#powerrail
      Contact( "Etapas_Grafcet".ETAPA_6 )
      wire#w1
      Contact( "Dados_Ciclo".FECHO_FILT_2 )
      wire#w2
      { S7_Templates := "SrcType := String" } NE_Contact(in1 := "Dados_Ciclo".POS_EVS_FILT_1, in2 := 'RINSE')
      wire#w3
      Contact( "T_POS_EVS".Q )
      wire#w5
      S_Coil( "Etapas_Grafcet".ETAPA_11 )
   END_RUNG
   RUNG wire#powerrail
      Contact( "Etapas_Grafcet".ETAPA_7 )
   END_RUNG wire#w1
   RUNG wire#powerrail
      Contact( "Etapas_Grafcet".ETAPA_8 )
   END_RUNG wire#w1
   RUNG wire#w2
      { S7_Templates := "SrcType := String" } NE_Contact(in1 := "Dados_Ciclo".POS_EVS_FILT_2, in2 := 'FECHO')
   END_RUNG wire#w3
   RUNG wire#w1
      Contact( "Dados_Ciclo".FECHO_FILT_1 )
      wire#w4
      { S7_Templates := "SrcType := String" } NE_Contact(in1 := "Dados_Ciclo".POS_EVS_FILT_1, in2 := 'FECHO')
   END_RUNG wire#w3
   RUNG wire#w4
      { S7_Templates := "SrcType := String" } NE_Contact(in1 := "Dados_Ciclo".POS_EVS_FILT_2, in2 := 'RINSE')
   END_RUNG wire#w3
   RUNG wire#w3
      Contact( "Etapas_Grafcet".ETAPA_7 )
   END_RUNG wire#w5
   RUNG wire#w3
      Contact( "Etapas_Grafcet".ETAPA_8 )
   END_RUNG wire#w5
   RUNG wire#w5
      R_Coil( "Etapas_Grafcet".ETAPA_6 )
   END_RUNG
   RUNG wire#w5
      R_Coil( "Etapas_Grafcet".ETAPA_7 )
   END_RUNG
   RUNG wire#w5
      R_Coil( "Etapas_Grafcet".ETAPA_8 )
   END_RUNG
   // the same network as SCL:
   IF ("Etapas_Grafcet".ETAPA_6 OR "Etapas_Grafcet".ETAPA_7 OR "Etapas_Grafcet".ETAPA_8) AND (("Dados_Ciclo".FECHO_FILT_2 AND (("Dados_Ciclo".POS_EVS_FILT_1 <> 'RINSE') OR ("Dados_Ciclo".POS_EVS_FILT_2 <> 'FECHO'))) OR ("Dados_Ciclo".FECHO_FILT_1 AND (("Dados_Ciclo".POS_EVS_FILT_1 <> 'FECHO') OR ("Dados_Ciclo".POS_EVS_FILT_2 <> 'RINSE')))) AND ("T_POS_EVS".Q OR "Etapas_Grafcet".ETAPA_7 OR "Etapas_Grafcet".ETAPA_8) THEN
       "Etapas_Grafcet".ETAPA_11 := TRUE;
   END_IF;
   #_w1 := ("Etapas_Grafcet".ETAPA_6 OR "Etapas_Grafcet".ETAPA_7 OR "Etapas_Grafcet".ETAPA_8) AND (("Dados_Ciclo".FECHO_FILT_2 AND (("Dados_Ciclo".POS_EVS_FILT_1 <> 'RINSE') OR ("Dados_Ciclo".POS_EVS_FILT_2 <> 'FECHO'))) OR ("Dados_Ciclo".FECHO_FILT_1 AND (("Dados_Ciclo".POS_EVS_FILT_1 <> 'FECHO') OR ("Dados_Ciclo".POS_EVS_FILT_2 <> 'RINSE')))) AND ("T_POS_EVS".Q OR "Etapas_Grafcet".ETAPA_7 OR "Etapas_Grafcet".ETAPA_8);
   IF #_w1 THEN
       "Etapas_Grafcet".ETAPA_6 := FALSE;
       "Etapas_Grafcet".ETAPA_7 := FALSE;
       "Etapas_Grafcet".ETAPA_8 := FALSE;
   END_IF;
END_REGION

REGION Network 12: ETAPA 12 (Alarme posição filtração)
   // As ev's não estão na posição de filtração nos 2 filtros
   RUNG wire#powerrail
      Contact( "Etapas_Grafcet".ETAPA_9 )
      wire#w1
      { S7_Templates := "SrcType := String" } NE_Contact(in1 := "Dados_Ciclo".POS_EVS_FILT_1, in2 := 'FILTRACAO')
      wire#w2
      Contact( "T_POS_EVS".Q )
      wire#w3
      S_Coil( "Etapas_Grafcet".ETAPA_12 )
   END_RUNG
   RUNG wire#powerrail
      Contact( "Etapas_Grafcet".ETAPA_1 )
   END_RUNG wire#w1
   RUNG wire#powerrail
      Contact( "Etapas_Grafcet".ETAPA_2 )
   END_RUNG wire#w1
   RUNG wire#w1
      { S7_Templates := "SrcType := String" } NE_Contact(in1 := "Dados_Ciclo".POS_EVS_FILT_2, in2 := 'FILTRACAO')
   END_RUNG wire#w2
   RUNG wire#w2
      Contact( "Etapas_Grafcet".ETAPA_1 )
   END_RUNG wire#w3
   RUNG wire#w2
      Contact( "Etapas_Grafcet".ETAPA_2 )
   END_RUNG wire#w3
   RUNG wire#w3
      R_Coil( "Etapas_Grafcet".ETAPA_9 )
   END_RUNG
   RUNG wire#w3
      R_Coil( "Etapas_Grafcet".ETAPA_1 )
   END_RUNG
   RUNG wire#w3
      R_Coil( "Etapas_Grafcet".ETAPA_2 )
   END_RUNG
   // the same network as SCL:
   IF ("Etapas_Grafcet".ETAPA_9 OR "Etapas_Grafcet".ETAPA_1 OR "Etapas_Grafcet".ETAPA_2) AND (("Dados_Ciclo".POS_EVS_FILT_1 <> 'FILTRACAO') OR ("Dados_Ciclo".POS_EVS_FILT_2 <> 'FILTRACAO')) AND ("T_POS_EVS".Q OR "Etapas_Grafcet".ETAPA_1 OR "Etapas_Grafcet".ETAPA_2) THEN
       "Etapas_Grafcet".ETAPA_12 := TRUE;
   END_IF;
   #_w1 := ("Etapas_Grafcet".ETAPA_9 OR "Etapas_Grafcet".ETAPA_1 OR "Etapas_Grafcet".ETAPA_2) AND (("Dados_Ciclo".POS_EVS_FILT_1 <> 'FILTRACAO') OR ("Dados_Ciclo".POS_EVS_FILT_2 <> 'FILTRACAO')) AND ("T_POS_EVS".Q OR "Etapas_Grafcet".ETAPA_1 OR "Etapas_Grafcet".ETAPA_2);
   IF #_w1 THEN
       "Etapas_Grafcet".ETAPA_9 := FALSE;
       "Etapas_Grafcet".ETAPA_1 := FALSE;
       "Etapas_Grafcet".ETAPA_2 := FALSE;
   END_IF;
END_REGION

REGION Network 13: Etapa 13 (Preparação para modo manual)
   // A etapa_n são as etapas de 1 a 9. A etapa 13 corresponde à preparação para entrada em manual. Param as bombas e mantém a posição das válvulas da etapa anterior. O reset às etapas de 1 a 9 é feito em Controlo_Ciclo_Manual
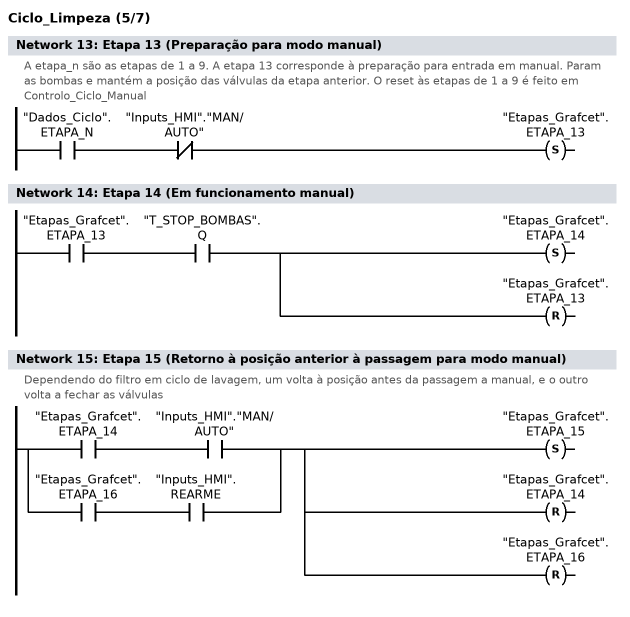
   RUNG wire#powerrail
      Contact( "Dados_Ciclo".ETAPA_N )
      I_Contact( "Inputs_HMI"."MAN/AUTO" )
      S_Coil( "Etapas_Grafcet".ETAPA_13 )
   END_RUNG
   // the same network as SCL:
   IF "Dados_Ciclo".ETAPA_N AND NOT "Inputs_HMI"."MAN/AUTO" THEN "Etapas_Grafcet".ETAPA_13 := TRUE; END_IF;
END_REGION

REGION Network 14: Etapa 14 (Em funcionamento manual)
   RUNG wire#powerrail
      Contact( "Etapas_Grafcet".ETAPA_13 )
      Contact( "T_STOP_BOMBAS".Q )
      wire#w1
      S_Coil( "Etapas_Grafcet".ETAPA_14 )
   END_RUNG
   RUNG wire#w1
      R_Coil( "Etapas_Grafcet".ETAPA_13 )
   END_RUNG
   // the same network as SCL:
   IF "Etapas_Grafcet".ETAPA_13 AND "T_STOP_BOMBAS".Q THEN
       "Etapas_Grafcet".ETAPA_14 := TRUE;
       "Etapas_Grafcet".ETAPA_13 := FALSE;
   END_IF;
END_REGION

REGION Network 15: Etapa 15 (Retorno à posição anterior à passagem para modo manual)
   // Dependendo do filtro em ciclo de lavagem, um volta à posição antes da passagem a manual, e o outro volta a fechar as válvulas
   RUNG wire#powerrail
      Contact( "Etapas_Grafcet".ETAPA_14 )
      Contact( "Inputs_HMI"."MAN/AUTO" )
      wire#w1
      S_Coil( "Etapas_Grafcet".ETAPA_15 )
   END_RUNG
   RUNG wire#powerrail
      Contact( "Etapas_Grafcet".ETAPA_16 )
      Contact( "Inputs_HMI".REARME )
   END_RUNG wire#w1
   RUNG wire#w1
      R_Coil( "Etapas_Grafcet".ETAPA_14 )
   END_RUNG
   RUNG wire#w1
      R_Coil( "Etapas_Grafcet".ETAPA_16 )
   END_RUNG
   // the same network as SCL:
   IF ("Etapas_Grafcet".ETAPA_14 AND "Inputs_HMI"."MAN/AUTO") OR ("Etapas_Grafcet".ETAPA_16 AND "Inputs_HMI".REARME) THEN
       "Etapas_Grafcet".ETAPA_15 := TRUE;
   END_IF;
   #_w1 := ("Etapas_Grafcet".ETAPA_14 AND "Inputs_HMI"."MAN/AUTO") OR ("Etapas_Grafcet".ETAPA_16 AND "Inputs_HMI".REARME);
   IF #_w1 THEN
       "Etapas_Grafcet".ETAPA_14 := FALSE;
       "Etapas_Grafcet".ETAPA_16 := FALSE;
   END_IF;
END_REGION

REGION Network 16: Etapa 16 (alarme em modo manual)
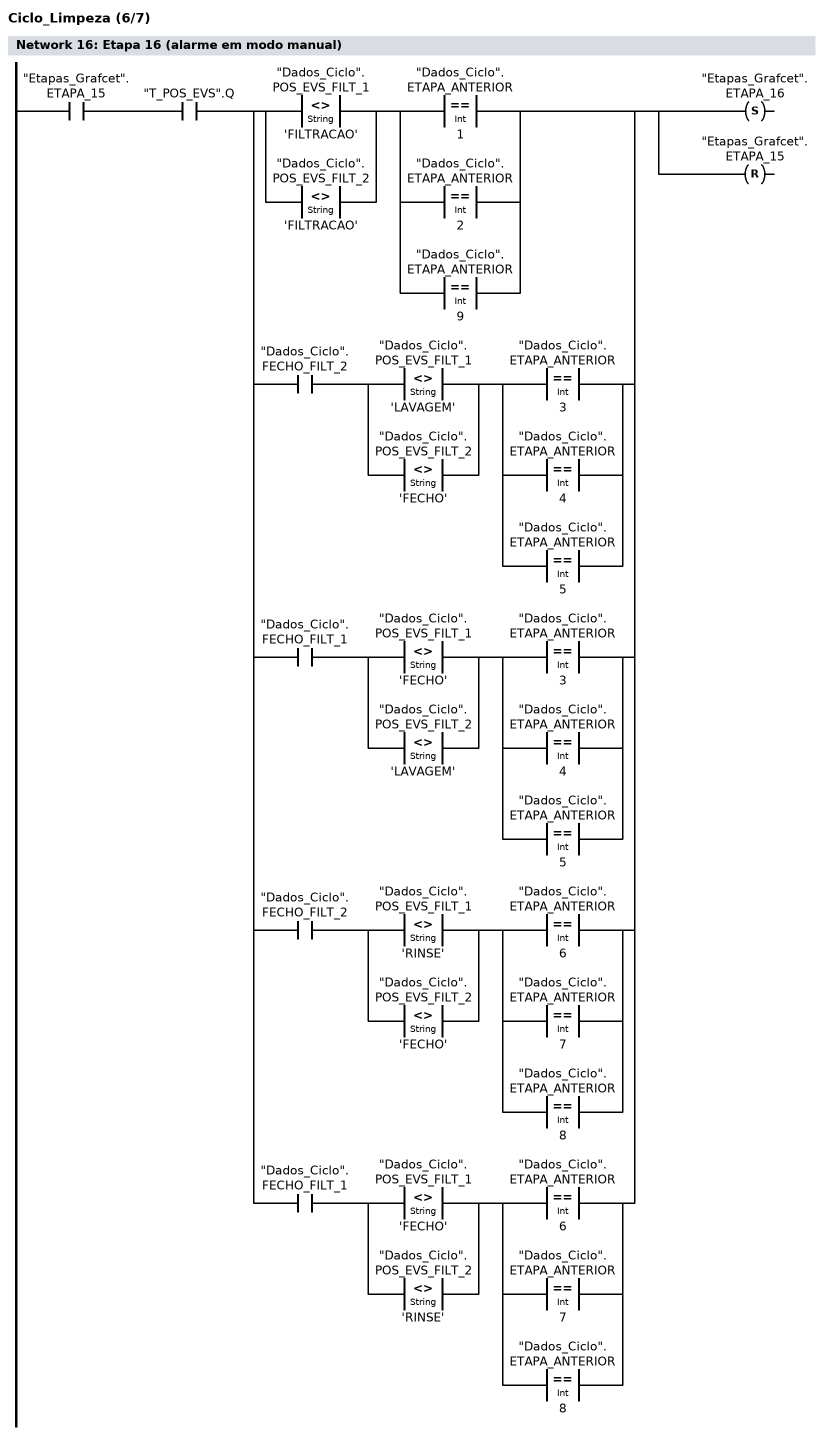
   RUNG wire#powerrail
      Contact( "Etapas_Grafcet".ETAPA_15 )
      Contact( "T_POS_EVS".Q )
      wire#w1
      { S7_Templates := "SrcType := String" } NE_Contact(in1 := "Dados_Ciclo".POS_EVS_FILT_1, in2 := 'FILTRACAO')
      wire#w2
      { S7_Templates := "SrcType := Int" } EQ_Contact(in1 := "Dados_Ciclo".ETAPA_ANTERIOR, in2 := 1)
      wire#w3
      S_Coil( "Etapas_Grafcet".ETAPA_16 )
   END_RUNG
   RUNG wire#w1
      { S7_Templates := "SrcType := String" } NE_Contact(in1 := "Dados_Ciclo".POS_EVS_FILT_2, in2 := 'FILTRACAO')
   END_RUNG wire#w2
   RUNG wire#w2
      { S7_Templates := "SrcType := Int" } EQ_Contact(in1 := "Dados_Ciclo".ETAPA_ANTERIOR, in2 := 2)
   END_RUNG wire#w3
   RUNG wire#w2
      { S7_Templates := "SrcType := Int" } EQ_Contact(in1 := "Dados_Ciclo".ETAPA_ANTERIOR, in2 := 9)
   END_RUNG wire#w3
   RUNG wire#w1
      Contact( "Dados_Ciclo".FECHO_FILT_2 )
      wire#w4
      { S7_Templates := "SrcType := String" } NE_Contact(in1 := "Dados_Ciclo".POS_EVS_FILT_1, in2 := 'LAVAGEM')
      wire#w5
      { S7_Templates := "SrcType := Int" } EQ_Contact(in1 := "Dados_Ciclo".ETAPA_ANTERIOR, in2 := 3)
   END_RUNG wire#w3
   RUNG wire#w4
      { S7_Templates := "SrcType := String" } NE_Contact(in1 := "Dados_Ciclo".POS_EVS_FILT_2, in2 := 'FECHO')
   END_RUNG wire#w5
   RUNG wire#w5
      { S7_Templates := "SrcType := Int" } EQ_Contact(in1 := "Dados_Ciclo".ETAPA_ANTERIOR, in2 := 4)
   END_RUNG wire#w3
   RUNG wire#w5
      { S7_Templates := "SrcType := Int" } EQ_Contact(in1 := "Dados_Ciclo".ETAPA_ANTERIOR, in2 := 5)
   END_RUNG wire#w3
   RUNG wire#w1
      Contact( "Dados_Ciclo".FECHO_FILT_1 )
      wire#w6
      { S7_Templates := "SrcType := String" } NE_Contact(in1 := "Dados_Ciclo".POS_EVS_FILT_1, in2 := 'FECHO')
      wire#w7
      { S7_Templates := "SrcType := Int" } EQ_Contact(in1 := "Dados_Ciclo".ETAPA_ANTERIOR, in2 := 3)
   END_RUNG wire#w3
   RUNG wire#w6
      { S7_Templates := "SrcType := String" } NE_Contact(in1 := "Dados_Ciclo".POS_EVS_FILT_2, in2 := 'LAVAGEM')
   END_RUNG wire#w7
   RUNG wire#w7
      { S7_Templates := "SrcType := Int" } EQ_Contact(in1 := "Dados_Ciclo".ETAPA_ANTERIOR, in2 := 4)
   END_RUNG wire#w3
   RUNG wire#w7
      { S7_Templates := "SrcType := Int" } EQ_Contact(in1 := "Dados_Ciclo".ETAPA_ANTERIOR, in2 := 5)
   END_RUNG wire#w3
   RUNG wire#w1
      Contact( "Dados_Ciclo".FECHO_FILT_2 )
      wire#w8
      { S7_Templates := "SrcType := String" } NE_Contact(in1 := "Dados_Ciclo".POS_EVS_FILT_1, in2 := 'RINSE')
      wire#w9
      { S7_Templates := "SrcType := Int" } EQ_Contact(in1 := "Dados_Ciclo".ETAPA_ANTERIOR, in2 := 6)
   END_RUNG wire#w3
   RUNG wire#w8
      { S7_Templates := "SrcType := String" } NE_Contact(in1 := "Dados_Ciclo".POS_EVS_FILT_2, in2 := 'FECHO')
   END_RUNG wire#w9
   RUNG wire#w9
      { S7_Templates := "SrcType := Int" } EQ_Contact(in1 := "Dados_Ciclo".ETAPA_ANTERIOR, in2 := 7)
   END_RUNG wire#w3
   RUNG wire#w9
      { S7_Templates := "SrcType := Int" } EQ_Contact(in1 := "Dados_Ciclo".ETAPA_ANTERIOR, in2 := 8)
   END_RUNG wire#w3
   RUNG wire#w1
      Contact( "Dados_Ciclo".FECHO_FILT_1 )
      wire#w10
      { S7_Templates := "SrcType := String" } NE_Contact(in1 := "Dados_Ciclo".POS_EVS_FILT_1, in2 := 'FECHO')
      wire#w11
      { S7_Templates := "SrcType := Int" } EQ_Contact(in1 := "Dados_Ciclo".ETAPA_ANTERIOR, in2 := 6)
   END_RUNG wire#w3
   RUNG wire#w10
      { S7_Templates := "SrcType := String" } NE_Contact(in1 := "Dados_Ciclo".POS_EVS_FILT_2, in2 := 'RINSE')
   END_RUNG wire#w11
   RUNG wire#w11
      { S7_Templates := "SrcType := Int" } EQ_Contact(in1 := "Dados_Ciclo".ETAPA_ANTERIOR, in2 := 7)
   END_RUNG wire#w3
   RUNG wire#w11
      { S7_Templates := "SrcType := Int" } EQ_Contact(in1 := "Dados_Ciclo".ETAPA_ANTERIOR, in2 := 8)
   END_RUNG wire#w3
   RUNG wire#w3
      R_Coil( "Etapas_Grafcet".ETAPA_15 )
   END_RUNG
   // the same network as SCL:
   IF "Etapas_Grafcet".ETAPA_15 AND "T_POS_EVS".Q AND (((("Dados_Ciclo".POS_EVS_FILT_1 <> 'FILTRACAO') OR ("Dados_Ciclo".POS_EVS_FILT_2 <> 'FILTRACAO')) AND (("Dados_Ciclo".ETAPA_ANTERIOR = 1) OR ("Dados_Ciclo".ETAPA_ANTERIOR = 2) OR ("Dados_Ciclo".ETAPA_ANTERIOR = 9))) OR ("Dados_Ciclo".FECHO_FILT_2 AND (("Dados_Ciclo".POS_EVS_FILT_1 <> 'LAVAGEM') OR ("Dados_Ciclo".POS_EVS_FILT_2 <> 'FECHO')) AND (("Dados_Ciclo".ETAPA_ANTERIOR = 3) OR ("Dados_Ciclo".ETAPA_ANTERIOR = 4) OR ("Dados_Ciclo".ETAPA_ANTERIOR = 5))) OR ("Dados_Ciclo".FECHO_FILT_1 AND (("Dados_Ciclo".POS_EVS_FILT_1 <> 'FECHO') OR ("Dados_Ciclo".POS_EVS_FILT_2 <> 'LAVAGEM')) AND (("Dados_Ciclo".ETAPA_ANTERIOR = 3) OR ("Dados_Ciclo".ETAPA_ANTERIOR = 4) OR ("Dados_Ciclo".ETAPA_ANTERIOR = 5))) OR ("Dados_Ciclo".FECHO_FILT_2 AND (("Dados_Ciclo".POS_EVS_FILT_1 <> 'RINSE') OR ("Dados_Ciclo".POS_EVS_FILT_2 <> 'FECHO')) AND (("Dados_Ciclo".ETAPA_ANTERIOR = 6) OR ("Dados_Ciclo".ETAPA_ANTERIOR = 7) OR ("Dados_Ciclo".ETAPA_ANTERIOR = 8))) OR ("Dados_Ciclo".FECHO_FILT_1 AND (("Dados_Ciclo".POS_EVS_FILT_1 <> 'FECHO') OR ("Dados_Ciclo".POS_EVS_FILT_2 <> 'RINSE')) AND (("Dados_Ciclo".ETAPA_ANTERIOR = 6) OR ("Dados_Ciclo".ETAPA_ANTERIOR = 7) OR ("Dados_Ciclo".ETAPA_ANTERIOR = 8)))) THEN
       "Etapas_Grafcet".ETAPA_16 := TRUE;
       "Etapas_Grafcet".ETAPA_15 := FALSE;
   END_IF;
END_REGION

REGION Network 17: Tempo de paragem das bombas (T1 no grafcet)
   // Espera um dado tempo para que as bombas parem, de modo a poder mudar a posição das ev's
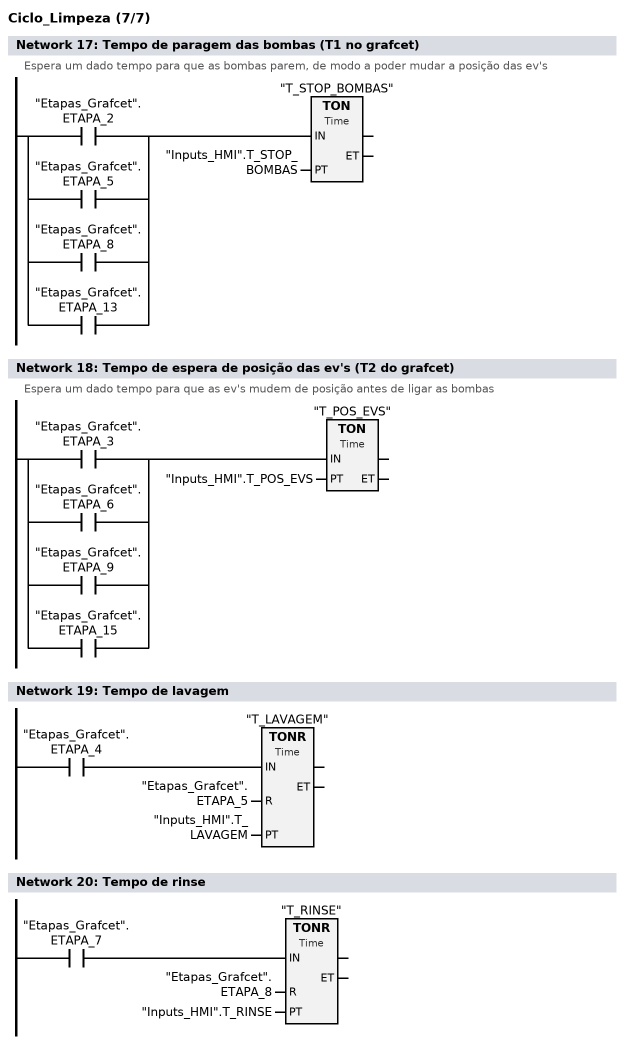
   RUNG wire#powerrail
      Contact( "Etapas_Grafcet".ETAPA_2 )
      wire#w1
      { S7_Templates := "time_type := Time" } "T_STOP_BOMBAS".TON(pt := "Inputs_HMI".T_STOP_BOMBAS, et =>)
   END_RUNG
   RUNG wire#powerrail
      Contact( "Etapas_Grafcet".ETAPA_5 )
   END_RUNG wire#w1
   RUNG wire#powerrail
      Contact( "Etapas_Grafcet".ETAPA_8 )
   END_RUNG wire#w1
   RUNG wire#powerrail
      Contact( "Etapas_Grafcet".ETAPA_13 )
   END_RUNG wire#w1
   // the same network as SCL:
   "T_STOP_BOMBAS".TON(IN := "Etapas_Grafcet".ETAPA_2 OR "Etapas_Grafcet".ETAPA_5 OR "Etapas_Grafcet".ETAPA_8 OR "Etapas_Grafcet".ETAPA_13,
                       PT := "Inputs_HMI".T_STOP_BOMBAS);
END_REGION

REGION Network 18: Tempo de espera de posição das ev's (T2 do grafcet)
   // Espera um dado tempo para que as ev's mudem de posição antes de ligar as bombas
   RUNG wire#powerrail
      Contact( "Etapas_Grafcet".ETAPA_3 )
      wire#w1
      { S7_Templates := "time_type := Time" } "T_POS_EVS".TON(pt := "Inputs_HMI".T_POS_EVS, et =>)
   END_RUNG
   RUNG wire#powerrail
      Contact( "Etapas_Grafcet".ETAPA_6 )
   END_RUNG wire#w1
   RUNG wire#powerrail
      Contact( "Etapas_Grafcet".ETAPA_9 )
   END_RUNG wire#w1
   RUNG wire#powerrail
      Contact( "Etapas_Grafcet".ETAPA_15 )
   END_RUNG wire#w1
   // the same network as SCL:
   "T_POS_EVS".TON(IN := "Etapas_Grafcet".ETAPA_3 OR "Etapas_Grafcet".ETAPA_6 OR "Etapas_Grafcet".ETAPA_9 OR "Etapas_Grafcet".ETAPA_15,
                   PT := "Inputs_HMI".T_POS_EVS);
END_REGION

REGION Network 19: Tempo de lavagem
   RUNG wire#powerrail
      Contact( "Etapas_Grafcet".ETAPA_4 )
      { S7_Templates := "time_type := Time" } "T_LAVAGEM".TONR(r := "Etapas_Grafcet".ETAPA_5, pt := "Inputs_HMI".T_LAVAGEM, et =>)
   END_RUNG
   // the same network as SCL:
   "T_LAVAGEM".TONR(IN := "Etapas_Grafcet".ETAPA_4, R := "Etapas_Grafcet".ETAPA_5, PT := "Inputs_HMI".T_LAVAGEM);
END_REGION

REGION Network 20: Tempo de rinse
   RUNG wire#powerrail
      Contact( "Etapas_Grafcet".ETAPA_7 )
      { S7_Templates := "time_type := Time" } "T_RINSE".TONR(r := "Etapas_Grafcet".ETAPA_8, pt := "Inputs_HMI".T_RINSE, et =>)
   END_RUNG
   // the same network as SCL:
   "T_RINSE".TONR(IN := "Etapas_Grafcet".ETAPA_7, R := "Etapas_Grafcet".ETAPA_8, PT := "Inputs_HMI".T_RINSE);
END_REGION
END_FUNCTION
